// TIA Portal V18 export
// export: Created 2025-12-01T12:39:35.2492762Z, ExportSetting None, DisplayName Totally Integrated Automation Portal, DisplayVersion V18 Update 5, DisplayName TIA Portal Openness, DisplayVersion V18 Update 5, DisplayName TIA Portal Teamcenter Gateway, DisplayVersion V18, DisplayName TIA Portal Version Control Interface, DisplayVersion V18, DisplayName STEP 7 Professional, DisplayVersion V18 Update 5, DisplayName STEP 7 Safety, DisplayVersion V18, DisplayName WinCC Professional, DisplayVersion V18 Update 5
VAR_GLOBAL   // PLC tag table "RemoteIO_DO_1"
   "oH-shaftLiftingLiftingCylinderToWP" AT %Q1000.0 : Bool;   // H-shaft 顶升位顶升气缸 去工作位
   "oH-shaftLiftingLiftingCylinderToHP" AT %Q1000.1 : Bool;   // H-shaft 顶升位顶升气缸 去原始位
   "oJ-magnetLiftingLiftingCylinderToWP" AT %Q1000.2 : Bool;   // J-magnet 顶升顶升气缸 去工作位
   "oJ-magnetLiftingLiftingCylinderToHP" AT %Q1000.3 : Bool;   // J-magnet 顶升顶升气缸 去原始位
   "oB-PressFitting-01GripperCylinderToWP" AT %Q1000.4 : Bool;   // B-压装模组-01夹爪气缸 去工作位
   "oB-PressFitting-01GripperCylinderToHP" AT %Q1000.5 : Bool;   // B-压装模组-01夹爪气缸 去原始位
   "oB-PressFitting-01CylinderToWP" AT %Q1000.6 : Bool;   // B-压装模组-01中转气缸 去工作位
   "oB-PressFitting-01CylinderToHP" AT %Q1000.7 : Bool;   // B-压装模组-01中转气缸 去原始位
   "oA-Loading-01HorizontalCylinderToWP" AT %Q1001.0 : Bool;   // A-转盘上料-01水平移栽气缸 去工作位
   "oA-Loading-01HorizontalCylinderToHP" AT %Q1001.1 : Bool;   // A-转盘上料-01水平移栽气缸 去原始位
   "oA-Loading-01UpDownTakeCylinderToWP" AT %Q1001.2 : Bool;   // A-转盘上料-01上下取料气缸 去工作位
   "oA-Loading-01UpDownTakeCylinderToHP" AT %Q1001.3 : Bool;   // A-转盘上料-01上下取料气缸 去原始位
   "oC-LocationCylinderToWP" AT %Q1001.4 : Bool;   // C-涂胶定位模组标准气缸 去工作位
   "oC-LocationCylinderToHP" AT %Q1001.5 : Bool;   // C-涂胶定位模组标准气缸 去原始位
   "oE-NG-01NGLocationCylinderToWP" AT %Q1001.6 : Bool;   // E-NG料盒-01NG定位气缸 去工作位
   "oE-NG-01NGLocationCylinderToHP" AT %Q1001.7 : Bool;   // E-NG料盒-01NG定位气缸 去原始位
   "oH-shaftLiftingPalletLocationCylinderToWP" AT %Q1002.0 : Bool;   // H-shaft 顶升位托盘定位气缸 去工作位
   "oH-shaftLiftingPalletLocationCylinderToHP" AT %Q1002.1 : Bool;   // H-shaft 顶升位托盘定位气缸 去原始位
   "oJ-magnetLiftingPalletLocationCylinderToWP" AT %Q1002.2 : Bool;   // J-magnet 顶升托盘定位气缸 去工作位
   "oJ-magnetLiftingPalletLocationCylinderToHP" AT %Q1002.3 : Bool;   // J-magnet 顶升托盘定位气缸 去原始位
   "RESERVE_Q1002.4" AT %Q1002.4 : Bool;   // 备用_Q1002.4
   "RESERVE_Q1002.5" AT %Q1002.5 : Bool;   // 备用_Q1002.5
   "RESERVE_Q1002.6" AT %Q1002.6 : Bool;   // 备用_Q1002.6
   "RESERVE_Q1002.7" AT %Q1002.7 : Bool;   // 备用_Q1002.7
   "oK-reserveLifting3LiftingCylinderToWP" AT %Q1006.0 : Bool;   // K-预留顶升位3顶升气缸 去工作位
   "oK-reserveLifting3LiftingCylinderToHP" AT %Q1006.1 : Bool;   // K-预留顶升位3顶升气缸 去原始位
   "oL-UnloadingTransCylinderToWP" AT %Q1006.2 : Bool;   // L-下料线体移栽气缸 去工作位
   "oL-UnloadingTransCylinderToHP" AT %Q1006.3 : Bool;   // L-下料线体移栽气缸 去原始位
   "oB-PressFitting-02GripperCylinderToWP" AT %Q1006.4 : Bool;   // B-压装模组-02夹爪气缸 去工作位
   "oB-PressFitting-02GripperCylinderToHP" AT %Q1006.5 : Bool;   // B-压装模组-02夹爪气缸 去原始位
   "oB-PressFitting-02CylinderToWP" AT %Q1006.6 : Bool;   // B-压装模组-02中转气缸 去工作位
   "oB-PressFitting-02CylinderToHP" AT %Q1006.7 : Bool;   // B-压装模组-02中转气缸 去原始位
   "oA-Loading-02HorizontalCylinderToWP" AT %Q1007.0 : Bool;   // A-转盘上料-02水平移栽气缸 去工作位
   "oA-Loading-02HorizontalCylinderToHP" AT %Q1007.1 : Bool;   // A-转盘上料-02水平移栽气缸 去原始位
   "oA-Loading-02UpDownTakeCylinderToWP" AT %Q1007.2 : Bool;   // A-转盘上料-02上下取料气缸 去工作位
   "oA-Loading-02UpDownTakeCylinderToHP" AT %Q1007.3 : Bool;   // A-转盘上料-02上下取料气缸 去原始位
   "oE-NG-02NGLocationCylinderToWP" AT %Q1007.4 : Bool;   // E-NG料盒-02NG定位气缸 去工作位
   "oE-NG-02NGLocationCylinderToHP" AT %Q1007.5 : Bool;   // E-NG料盒-02NG定位气缸 去原始位
   "oK-reserveLifting3PalletLocationCylinderToWP" AT %Q1007.6 : Bool;   // K-预留顶升位3托盘定位气缸 去工作位
   "oK-reserveLifting3PalletLocationCylinderToHP" AT %Q1007.7 : Bool;   // K-预留顶升位3托盘定位气缸 去原始位
   "oL-UnloadingTransPalletLocationCylinderToWP" AT %Q1008.0 : Bool;   // L-下料线体移栽托盘定位气缸 去工作位
   "oL-UnloadingTransPalletLocationCylinderToHP" AT %Q1008.1 : Bool;   // L-下料线体移栽托盘定位气缸 去原始位
   "RESERVE_Q1008.2" AT %Q1008.2 : Bool;
   "RESERVE_Q1008.3" AT %Q1008.3 : Bool;
   "RESERVE_Q1008.4" AT %Q1008.4 : Bool;
   "RESERVE_Q1008.5" AT %Q1008.5 : Bool;
   "RESERVE_Q1008.6" AT %Q1008.6 : Bool;
   "RESERVE_Q1008.7" AT %Q1008.7 : Bool;
   "oF-ROOBT1Gripper1CylinderToWP" AT %Q1100.0 : Bool;   // F-ROBOT 1夹爪1夹爪气缸 去工作位
   "oF-ROOBT1Gripper1CylinderToHP" AT %Q1100.1 : Bool;   // F-ROBOT 1夹爪1夹爪气缸 去原始位
   "oF-ROOBT1Gripper2CylinderToWP" AT %Q1100.2 : Bool;   // F-ROBOT 1夹爪2夹爪气缸 去工作位
   "oF-ROOBT1Gripper2CylinderToHP" AT %Q1100.3 : Bool;   // F-ROBOT 1夹爪2夹爪气缸 去原始位
   "RESERVE_Q1100.4" AT %Q1100.4 : Bool;   // 备用_Q1100.4
   "RESERVE_Q1100.5" AT %Q1100.5 : Bool;   // 备用_Q1100.5
   "RESERVE_Q1100.6" AT %Q1100.6 : Bool;   // 备用_Q1100.6
   "RESERVE_Q1100.7" AT %Q1100.7 : Bool;   // 备用_Q1100.7
   "oF-ROOBT2Gripper1CylinderToWP" AT %Q1102.0 : Bool;   // F-ROBOT2夹爪1夹爪气缸 去工作位
   "oF-ROOBT2Gripper1CylinderToHP" AT %Q1102.1 : Bool;   // F-ROBOT2夹爪1夹爪气缸 去原始位
   "oF-ROOBT2Gripper2CylinderToWP" AT %Q1102.2 : Bool;   // F-ROBOT2夹爪2夹爪气缸 去工作位
   "oF-ROOBT2Gripper2CylinderToHP" AT %Q1102.3 : Bool;   // F-ROBOT2夹爪2夹爪气缸 去原始位
   "RESERVE_Q1102.4" AT %Q1102.4 : Bool;   // 备用_Q1102.4
   "RESERVE_Q1102.5" AT %Q1102.5 : Bool;   // 备用_Q1102.5
   "RESERVE_Q1102.6" AT %Q1102.6 : Bool;   // 备用_Q1102.6
   "RESERVE_Q1102.7" AT %Q1102.7 : Bool;   // 备用_Q1102.7
   "oF-ROOBT3Gripper1CylinderToWP" AT %Q1104.0 : Bool;   // F-ROBOT 3夹爪1夹爪气缸 去工作位
   "oF-ROOBT3Gripper1CylinderToHP" AT %Q1104.1 : Bool;   // F-ROBOT 3夹爪1夹爪气缸 去原始位
   "oF-ROOBT3Gripper2CylinderToWP" AT %Q1104.2 : Bool;   // F-ROBOT 3夹爪2夹爪气缸 去工作位
   "oF-ROOBT3Gripper2CylinderToHP" AT %Q1104.3 : Bool;   // F-ROBOT 3夹爪2夹爪气缸 去原始位
   "RESERVE_Q1104.4" AT %Q1104.4 : Bool;   // 备用_Q1104.4
   "RESERVE_Q1104.5" AT %Q1104.5 : Bool;   // 备用_Q1104.5
   "RESERVE_Q1104.6" AT %Q1104.6 : Bool;   // 备用_Q1104.6
   "RESERVE_Q1104.7" AT %Q1104.7 : Bool;   // 备用_Q1104.7
END_VAR
